(* PLC project FromServer, Turbopneumatic Socket Server 1, author DVorobiev *)
(* stored: creationDateTime 2020-11-19T10:39:58, productRelease 1, companyURL www.turbo.ru, modificationDateTime 2020-12-04T16:33:17, version 1, organization Turbopneumatic *)

(* mainServer *)
PROGRAM mainServer1
  VAR
    python_eval0 : python_eval;
    trigger : BOOL := False;
    trigger0 : BOOL := False;
    s_out : STRING;
    d_value : LREAL;
    python_eval1 : python_eval;
  END_VAR
  VAR  (* added by the conversion: wires and edge detectors of the diagram *)
    _NOT8_OUT : BOOL;
    _NOT4_OUT : BOOL;
  END_VAR

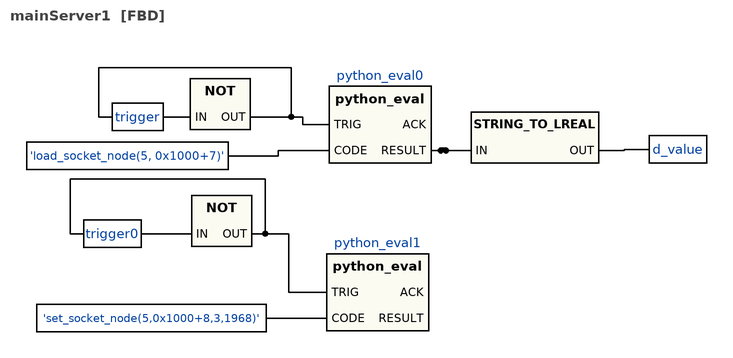
(* FBD diagram, written out as Structured Text *)
_NOT8_OUT := NOT trigger;
trigger := _NOT8_OUT;
python_eval0(TRIG := _NOT8_OUT, CODE := 'load_socket_node(5, 0x1000+7)');
d_value := STRING_TO_LREAL(python_eval0.RESULT);
_NOT4_OUT := NOT trigger0;
trigger0 := _NOT4_OUT;
python_eval1(TRIG := _NOT4_OUT, CODE := 'set_socket_node(5,0x1000+8,3,1968)');
END_PROGRAM

(* load_socket_node parameters *)
FUNCTION set_load_param : STRING
  VAR_INPUT
    id_Node : INT;
    id_Obj : INT;
    id_SubObj : INT;
  END_VAR

            set_load_param:=CONCAT('load_socket_node(',INT_TO_STRING(id_Node),',',INT_TO_STRING(id_Obj),')');


          
END_FUNCTION

(* Loading information from Node *)
FUNCTION_BLOCK load_socket_node
  VAR
    pyTrigger : BOOL;
  END_VAR
  VAR_INPUT
    id_Node : INT := 1;  (* Id for Node *)
    id_Obj : INT := 4096;  (* Id for Obj *)
    id_SubObj : INT := 0;  (* Id for SubObj *)
  END_VAR
  VAR
    python_eval0 : python_eval;
  END_VAR
  VAR_OUTPUT
    d_value : LREAL;
  END_VAR
  VAR  (* added by the conversion: wires and edge detectors of the diagram *)
    _NOT2_OUT : BOOL;
  END_VAR

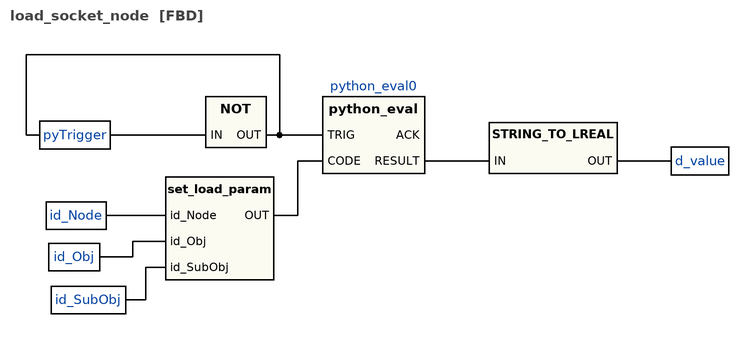
(* FBD diagram, written out as Structured Text *)
_NOT2_OUT := NOT pyTrigger;
pyTrigger := _NOT2_OUT;
python_eval0(TRIG := _NOT2_OUT, CODE := set_load_param(id_Node, id_Obj, id_SubObj));
d_value := STRING_TO_LREAL(python_eval0.RESULT);
END_FUNCTION_BLOCK

(* mainServer *)
PROGRAM mainServer
  VAR
    id_Node : INT := 5;
    i_Obj : INT := 4103;
    i_SubObj : INT := 0;
    trigger0 : BOOL := False;
    s_out : STRING;
    d_value : LREAL;
    d_val_out_1 : REAL;
    python_eval1 : python_eval;
    load_socket_node0 : load_socket_node;
    INTEGRAL0 : INTEGRAL;
    cycle : STRING := '0:0:1';
  END_VAR
  VAR  (* added by the conversion: wires and edge detectors of the diagram *)
    _NOT14_OUT : BOOL;
  END_VAR

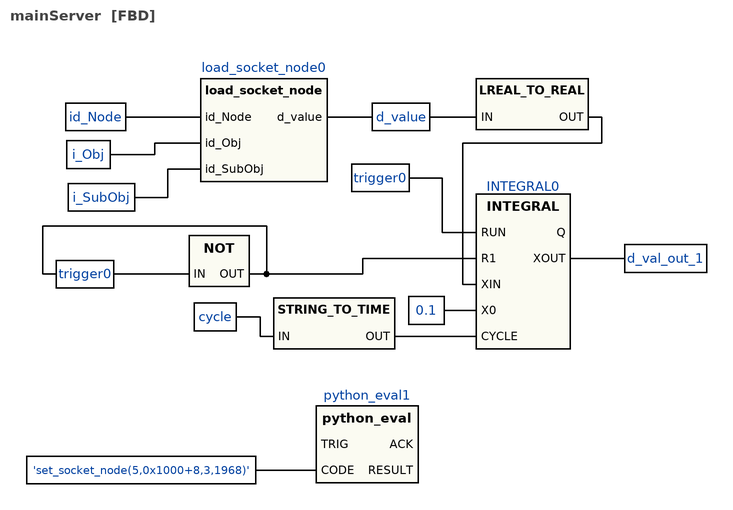
(* FBD diagram, written out as Structured Text *)
load_socket_node0(id_Node := id_Node, id_Obj := i_Obj, id_SubObj := i_SubObj);
d_value := load_socket_node0.d_value;
_NOT14_OUT := NOT trigger0;
INTEGRAL0(RUN := trigger0, R1 := _NOT14_OUT, XIN := LREAL_TO_REAL(d_value), X0 := 0.1, CYCLE := STRING_TO_TIME(cycle));
d_val_out_1 := INTEGRAL0.XOUT;
trigger0 := _NOT14_OUT;
python_eval1(CODE := 'set_socket_node(5,0x1000+8,3,1968)');
END_PROGRAM

CONFIGURATION config
  RESOURCE resource1 ON PLC
    TASK taskServer(INTERVAL := T#1s0ms, PRIORITY := 0);
    PROGRAM srv WITH taskServer : mainServer;
  END_RESOURCE
END_CONFIGURATION
